(* PLC project Tc2_Utilities.FB_EnumStringNumbers Demo, tc3-libraries-kb TwinCAT 3.1 *)
(* stored: creationDateTime 2026-05-10T20:00:00, modificationDateTime 2026-05-10T20:00:00 *)

PROGRAM P_Demo_FB_EnumStringNumbers
  VAR
    fbFB_EnumStringNumbers : FB_EnumStringNumbers;  (* Tc2_Utilities.FB_EnumStringNumbers 实例 *)
    arg_sSearch : T_MaxString;  (* VAR_INPUT sSearch *)
    arg_eCmd : E_EnumCmdType;  (* VAR_INPUT eCmd *)
    arg_eType : E_NumGroupTypes;  (* VAR_INPUT eType *)
    out_sNumber : T_MaxString;  (* VAR_OUTPUT sNumber *)
    out_nPos : INT;  (* VAR_OUTPUT nPos *)
    out_bEOS : BOOL;  (* VAR_OUTPUT bEOS *)
  END_VAR

            // ============================================================
// Tc2_Utilities.FB_EnumStringNumbers 演示程序（FB 实例）
// ============================================================
// 验证步骤：
//   1. 引用 Tc2_Utilities（及依赖类型所在库 Tc2_System 等）
//   2. 编译 + 登录
//   3. 按 doc.md 给 arg_* 赋值
//   4. 在线监视 out_* / io_* 输出
// ============================================================

fbFB_EnumStringNumbers(
    sSearch := arg_sSearch,
    eCmd := arg_eCmd,
    eType := arg_eType,
    sNumber => out_sNumber,
    nPos => out_nPos,
    bEOS => out_bEOS
);

          
END_PROGRAM
